(* PLC project prj, KAIST_DSLAB noNameNow 1, author bwkim *)
(* stored: creationDateTime 2012-2-3T08:19:06, modificationDateTime 2012-2-3T08:19:06 *)

FUNCTION_BLOCK OR
  VAR_INPUT
    A : BOOL := FALSE;
  END_VAR
  VAR_INPUT
    B : BOOL := FALSE;
  END_VAR
  VAR_INPUT
    C : BOOL := FALSE;
  END_VAR
  VAR_INPUT
    _D : BOOL := FALSE;
  END_VAR
  VAR_OUTPUT
    OR4 : BOOL := FALSE;
  END_VAR

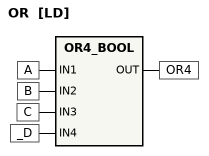
(* LD diagram, written out as Structured Text *)
OR4 := OR4_BOOL(A, B, C, _D);
END_FUNCTION_BLOCK
